PROGRAM MAIN
VAR
	fbSerialCommunication 			: FB_SerialCommunication(nDatabits := 8, eParity := E_Parity.Even, nStopbits := 1);
	fbSerialCommunicationRS232 		: FB_SerialCommunicationRS232(nDatabits := 8, eParity := E_Parity.Even, nStopbits := 1, nBaudrate := 19200);	
	fbSerialCommunicationCluster	: FB_SerialCommunicationCluster(nDatabits := 8, eParity := E_Parity.None, nStopbits := 1);
END_VAR

fbSerialCommunication();
fbSerialCommunicationRS232();
fbSerialCommunicationCluster();

END_PROGRAM

(* stored: Version 1.1.0.1, ProductVersion 3.1.4024.0
   POU MAIN: Id {50728c29-9f9a-46da-ad77-0bcd7412a99c}, SpecialFunc None *)
